(* 
:Description: This function block is used to buffer all data base on FIFO concept.
*)
FUNCTION_BLOCK FB_DataSetFifo
VAR
	MAX_BUFFER_SIZE : UINT;
	arrBuffer 	: ARRAY[0..1000] OF BYTE; (* Buffer memory used by FB_MemRingBuffer function block *)
	fbBuffer	: FB_MemRingBuffer;
	
	_bOk		: BOOL;
	_nCount		: UDINT;
	_nLoad		: UDINT;
	_bOverwrite	: BOOL;
END_VAR

(*
Version history:

+-------------+------------+----------------+----------+------------------------------------------------------------+
|Date         | Version    | created under  | Author   | Remark                                                     |
+=============+============+================+==========+============================================================+
|2024-02      | 1.0.0.0    | V3.1.4024.22   | HVAP     | Function block created                                     |
+-------------+------------+----------------+----------+------------------------------------------------------------+

*)

;

METHOD AddData : BOOL
VAR_INPUT
	in : REAL;
END_VAR
fbBuffer.A_AddTail( pWrite:= ADR( in ),
					cbWrite:= SIZEOF( in ),
					pBuffer:= ADR( arrBuffer ),
					cbBuffer:= SIZEOF( arrBuffer ),
					bOk=> _bOk,
					nCount => _nCount );


IF NOT _bOk THEN (* overflow ? *)
	IF bOverwrite THEN
		fbBuffer.A_RemoveHead(); (* remove one oldest entry *)

		fbBuffer.A_AddTail( bOk => _bOk, nCount => _nCount );
	END_IF
END_IF



_nLoad := (fbBuffer.cbSize * 100) / 1000;
END_METHOD

PROPERTY Count : UDINT
GET
Count := _nCount;
END_GET
END_PROPERTY

METHOD GetData : BOOL
VAR_OUTPUT
	out : REAL;
END_VAR
fbBuffer.A_GetHead( pRead:= ADR( out ),
					cbRead:= SIZEOF( out ),
					pBuffer:= ADR( arrBuffer ),
					cbBuffer:= SIZEOF( arrBuffer ),
					bOk=> _bOk,
					nCount => _nCount );

_nLoad := (fbBuffer.cbSize * 100) / 1000;
END_METHOD

PROPERTY Load : UDINT
GET
Load := _nLoad;
END_GET
END_PROPERTY

PROPERTY OK : BOOL
GET
OK := _bOk;
END_GET
END_PROPERTY

PROPERTY OverWrite : BOOL
SET
_bOverwrite := OverWrite;
END_SET
END_PROPERTY

METHOD Remove : BOOL
VAR_OUTPUT
	out : REAL;
END_VAR
fbBuffer.A_RemoveHead( 	pRead:= ADR( out ),
						cbRead:= SIZEOF( out ),
						pBuffer:= ADR( arrBuffer ),
						cbBuffer:= SIZEOF( arrBuffer ),
						bOk=> _bOk,
						nCount => _nCount );

_nLoad := (fbBuffer.cbSize * 100) / 1000;
END_METHOD

METHOD Reset : BOOL
VAR_INPUT
END_VAR
MEMSET( ADR( arrBuffer ), 0, SIZEOF( arrBuffer ) ); (* reset (optional) internal buffer *)

fbBuffer.A_Reset( 	bOk=> _bOk,
					nCount => _nCount );

_nLoad := (fbBuffer.cbSize * 100) / 1000;
END_METHOD

END_FUNCTION_BLOCK

(* stored: Version 1.1.0.1, ProductVersion 3.1.4024.9
   POU FB_DataSetFifo: Id {68aab722-1c15-4a1c-8558-70d8155fb516}, SpecialFunc None
   Method AddData: Id {806cf257-e082-4499-824e-d35c7ee27f3b}
   Property Count: Id {42270d8d-a9c8-4f05-bae7-28d0249ec709}
   Get Get: Id {adb7774c-93a8-40e4-aac2-a9fa76af383e}
   Method GetData: Id {0e79a6b7-8e40-429c-beb1-e3e03e706085}
   Property Load: Id {6e073599-055b-4e4c-8496-d76ae7262bdd}
   Get Get: Id {b6fc64b1-9500-4ddf-a7bf-278fea2ae343}
   Property OK: Id {7fbf5742-1e65-42d7-a9a4-cbff4411ba3c}
   Get Get: Id {ab850ee0-1094-4d02-8af9-56e6be495ffe}
   Property OverWrite: Id {a4ded3f2-b8eb-4d1e-8863-706bacfdf317}
   Set Set: Id {efc885fc-c103-4190-8eaa-3578c12692a0}
   Method Remove: Id {ba69501a-1e41-46ca-9a82-0a3e70bd1fc2}
   Method Reset: Id {0c386d56-72f5-42dd-8228-c15774d39af4} *)
